// TIA Portal project "ProjectFESTO" (V15.1)

(* hardware
DEVICE "S7-1200 station_1"  S7-1200 Station
   slot 0: "Rack_0"  S7-1200 Rack  Rack  V1.0
   slot 1: "Distribution"  CPU 1214C DC/DC/DC  6ES7 214-1AG40-0XB0  V4.2
   slot 2: "DI 8/DQ 8x24VDC_1"  6ES7 223-1BH32-0XB0  V2.0
   slot 3: "SM 1278_1"  4SI IO link  6ES7 278-4BD32-0XB0  V2.1
DEVICE "S7-1200 station_2"  S7-1200 Station
   slot 0: "Rack_0"  S7-1200 Rack  Rack  V1.0
   slot 1: "Separation"  CPU 1214C DC/DC/DC  6ES7 214-1AG40-0XB0  V4.2
   slot 2: "DI 8/DQ 8x24VDC_1"  6ES7 223-1BH32-0XB0  V2.0
   slot 3: "SM 1278_1"  4SI IO link  6ES7 278-4BD32-0XB0  V2.1
*)

// ===== PLC "Distribution"  CPU 1214C DC/DC/DC =====

VAR_GLOBAL   // PLC tag table "DistributionIO"
   "WorkpieceAtBeginning" AT %I0.0 : Bool;
   "WorkpieceAtMiddle" AT %I0.1 : Bool;
   "NoWorkpieceAtEnd" AT %I0.2 : Bool;
   "SlideRetracted" AT %I0.4 : Bool;
   "SlideAdvanced" AT %I0.5 : Bool;
   "MagazineEmpty" AT %I0.6 : Bool;
   "ConveyorForward" AT %Q0.0 : Bool;
   "ConveyorReverse" AT %Q0.1 : Bool;
   "AdvanceFeedSeparator" AT %Q0.2 : Bool;
   "AdvanceSlide" AT %Q0.4 : Bool;
   "GreenButtonOn" AT %I8.0 : Bool;
   "RedButtonOff" AT %I8.1 : Bool;
   "Key" AT %I8.2 : Bool;
   "GrayButtonOn" AT %I8.3 : Bool;
   "SeparationDisponible" AT %I8.7 : Bool;
   "DistributionDisponible" AT %Q8.7 : Bool;
END_VAR

VAR_GLOBAL   // PLC tag table "DistributionMemory"
   "StateWorkpieceAtMagazine" AT %M0.0 : Bool;
   "StateWorkpieceAtConveyor" AT %M0.1 : Bool;
   "MoveToSeparation" AT %M0.2 : Bool;
END_VAR

ORGANIZATION_BLOCK "Main"   // OB1, LAD, ProgramCycle
TITLE = "Main Program Sweep (Cycle)"
{ S7_Optimized_Access := 'TRUE' }
VERSION : 0.1
   VAR_INPUT
      Initial_Call : Bool;   // Initial call of this OB
      Remanence : Bool;   // =True, if remanent data are available
   END_VAR
BEGIN

REGION Network 1
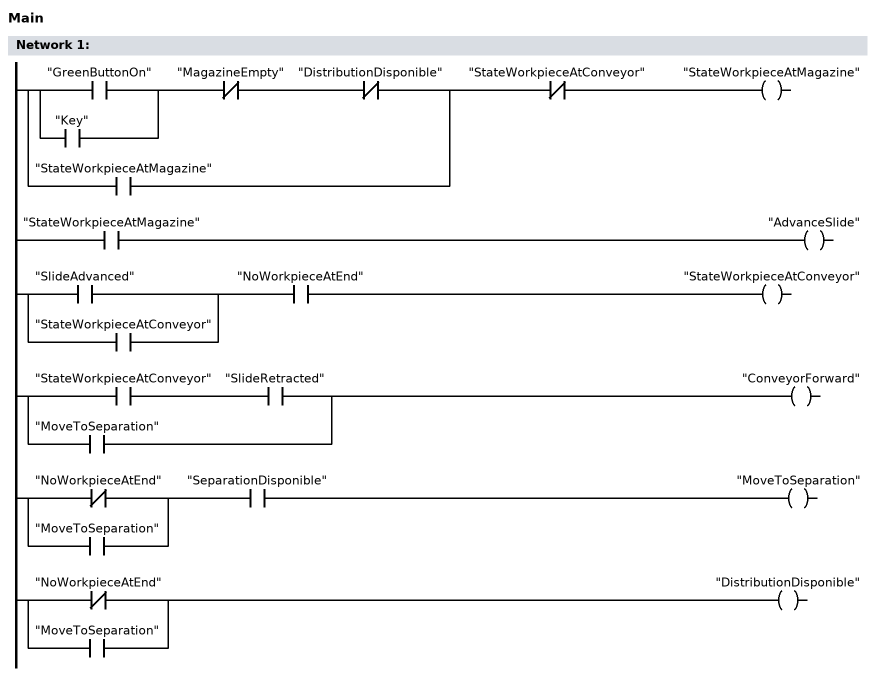
   RUNG wire#powerrail
      Contact( "GreenButtonOn" )
      wire#w1
      I_Contact( "MagazineEmpty" )
      I_Contact( "DistributionDisponible" )
      wire#w2
      I_Contact( "StateWorkpieceAtConveyor" )
      Coil( "StateWorkpieceAtMagazine" )
   END_RUNG
   RUNG wire#powerrail
      Contact( "Key" )
   END_RUNG wire#w1
   RUNG wire#powerrail
      Contact( "StateWorkpieceAtMagazine" )
   END_RUNG wire#w2
   RUNG wire#powerrail
      Contact( "StateWorkpieceAtMagazine" )
      Coil( "AdvanceSlide" )
   END_RUNG
   RUNG wire#powerrail
      Contact( "SlideAdvanced" )
      wire#w3
      Contact( "NoWorkpieceAtEnd" )
      Coil( "StateWorkpieceAtConveyor" )
   END_RUNG
   RUNG wire#powerrail
      Contact( "StateWorkpieceAtConveyor" )
   END_RUNG wire#w3
   RUNG wire#powerrail
      Contact( "StateWorkpieceAtConveyor" )
      Contact( "SlideRetracted" )
      wire#w4
      Coil( "ConveyorForward" )
   END_RUNG
   RUNG wire#powerrail
      Contact( "MoveToSeparation" )
   END_RUNG wire#w4
   RUNG wire#powerrail
      I_Contact( "NoWorkpieceAtEnd" )
      wire#w5
      Contact( "SeparationDisponible" )
      Coil( "MoveToSeparation" )
   END_RUNG
   RUNG wire#powerrail
      Contact( "MoveToSeparation" )
   END_RUNG wire#w5
   RUNG wire#powerrail
      I_Contact( "NoWorkpieceAtEnd" )
      wire#w6
      Coil( "DistributionDisponible" )
   END_RUNG
   RUNG wire#powerrail
      Contact( "MoveToSeparation" )
   END_RUNG wire#w6
   // the same network as SCL:
   "StateWorkpieceAtMagazine" := ((("GreenButtonOn" OR "Key") AND NOT "MagazineEmpty" AND NOT "DistributionDisponible") OR "StateWorkpieceAtMagazine") AND NOT "StateWorkpieceAtConveyor";
   "AdvanceSlide" := "StateWorkpieceAtMagazine";
   "StateWorkpieceAtConveyor" := ("SlideAdvanced" OR "StateWorkpieceAtConveyor") AND "NoWorkpieceAtEnd";
   "ConveyorForward" := ("StateWorkpieceAtConveyor" AND "SlideRetracted") OR "MoveToSeparation";
   "MoveToSeparation" := (NOT "NoWorkpieceAtEnd" OR "MoveToSeparation") AND "SeparationDisponible";
   "DistributionDisponible" := NOT "NoWorkpieceAtEnd" OR "MoveToSeparation";
END_REGION
END_ORGANIZATION_BLOCK

// ===== PLC "Separation"  CPU 1214C DC/DC/DC =====

VAR_GLOBAL   // PLC tag table "SeparationIO"
   "WorkpieceAtBeginning" AT %I0.0 : Bool;
   "Deflector1Extended" AT %I0.1 : Bool;
   "ChuteFull" AT %I0.2 : Bool;
   "Deflector2Extended" AT %I0.3 : Bool;
   "WorkpieceDetected" AT %I0.4 : Bool;
   "WorkpieceNotBlack" AT %I0.5 : Bool;
   "WorkpieceMetallic" AT %I0.6 : Bool;
   "ConveyorForward" AT %Q0.0 : Bool;
   "ExtendDeflector1" AT %Q0.1 : Bool;
   "ExtendDeflector2" AT %Q0.2 : Bool;
   "RetractStopper" AT %Q0.3 : Bool;
   "GreenButtonOn" AT %I8.0 : Bool;
   "RedButtonOff" AT %I8.1 : Bool;
   "Key" AT %I8.2 : Bool;
   "GrayButtonOn" AT %I8.3 : Bool;
   "SeparationDisponible" AT %Q8.5 : Bool;
   "DistributionDisponible" AT %I8.5 : Bool;
END_VAR

VAR_GLOBAL   // PLC tag table "SeparationMemory"
   "StateWorkpieceAtConveyor" AT %M0.0 : Bool;
   "StateWorkpieceSeparation" AT %M0.1 : Bool;
END_VAR

// folder: System blocks/Program resources

DATA_BLOCK "IEC_Timer_0_DB"   // DB1
{ S7_Optimized_Access := 'TRUE' }
AUTHOR : Simatic
FAMILY : IEC
NAME : IEC_TMR
VERSION : 1.0
// stored: InstanceOfName IEC_TIMER
"IEC_TIMER"
BEGIN
END_DATA_BLOCK

// folder: (top level)

ORGANIZATION_BLOCK "Main"   // OB1, LAD, ProgramCycle
TITLE = "Main Program Sweep (Cycle)"
{ S7_Optimized_Access := 'TRUE' }
VERSION : 0.1
   VAR_INPUT
      Initial_Call : Bool;   // Initial call of this OB
      Remanence : Bool;   // =True, if remanent data are available
   END_VAR
BEGIN

REGION Network 1
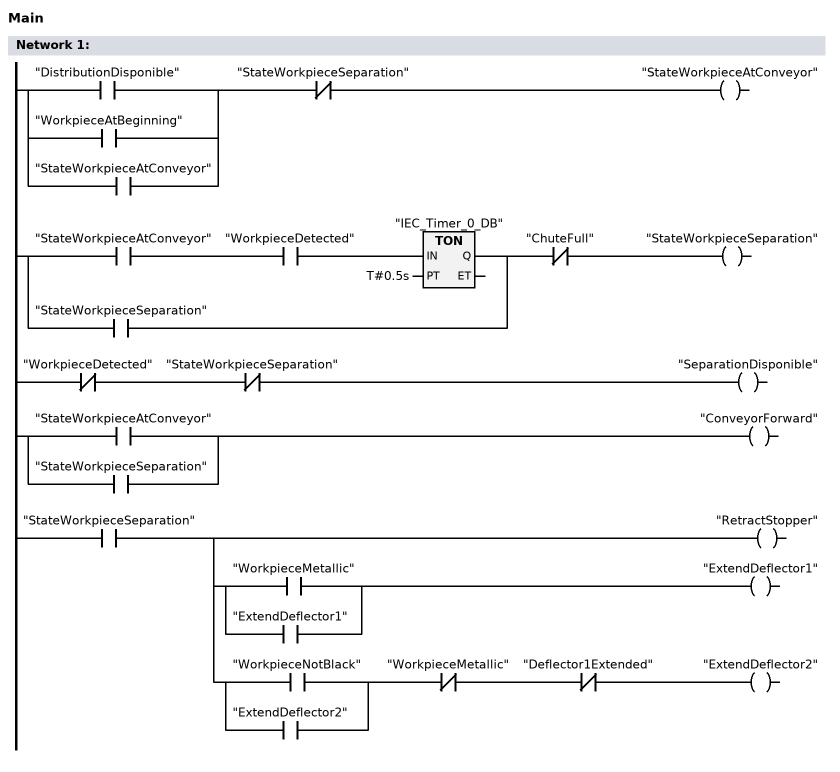
   "StateWorkpieceAtConveyor" := ("DistributionDisponible" OR "WorkpieceAtBeginning" OR "StateWorkpieceAtConveyor") AND NOT "StateWorkpieceSeparation";
   "IEC_Timer_0_DB".TON(IN := "StateWorkpieceAtConveyor" AND "WorkpieceDetected", PT := T#0.5s);
   "StateWorkpieceSeparation" := ("IEC_Timer_0_DB".Q OR "StateWorkpieceSeparation") AND NOT "ChuteFull";
   "SeparationDisponible" := NOT "WorkpieceDetected" AND NOT "StateWorkpieceSeparation";
   "ConveyorForward" := "StateWorkpieceAtConveyor" OR "StateWorkpieceSeparation";
   "RetractStopper" := "StateWorkpieceSeparation";
   "ExtendDeflector1" := "StateWorkpieceSeparation" AND ("WorkpieceMetallic" OR "ExtendDeflector1");
   "ExtendDeflector2" := "StateWorkpieceSeparation" AND ("WorkpieceNotBlack" OR "ExtendDeflector2") AND NOT "WorkpieceMetallic" AND NOT "Deflector1Extended";
END_REGION
END_ORGANIZATION_BLOCK